// Mitsubishi GX Works2 project: project_PLC_Final   PLC: FX3G

// global labels: Global1
VAR_GLOBAL
  start_switch AT X007 : BOOL;
END_VAR
VAR_GLOBAL CONSTANT
  reset : REAL;
END_VAR
VAR_GLOBAL
  chocolate_stock AT D2000 : REAL;
  nuts_stock AT D2400 : REAL;
  pistachio_stock AT D2800 : REAL;
  kadaif_stock AT D3200 : REAL;
  chocolate_input AT D2200 : REAL;
  nuts_input AT D2600 : REAL;
  pistachio_input AT D3000 : REAL;
  kadaif_input AT D3400 : REAL;
END_VAR
VAR_GLOBAL CONSTANT
  melting_chocolate : REAL := 400;
  mix_nuts : REAL := 100;
  dubai_package : REAL := 120;
  mix_nuts_packge : REAL := 100;
  kadaif_dubai_package : REAL := 60;
END_VAR
VAR_GLOBAL
  m_28 AT M28 : BOOL;
  m_27 AT M27 : BOOL;
  m_26 AT M26 : BOOL;
  m_25 AT M25 : BOOL;
  m_29 AT M29 : BOOL;
  m_30 AT M30 : BOOL;
  m_31 AT M31 : BOOL;
  m_32 AT M32 : BOOL;
  valid_input AT M153 : BOOL;
  active_day AT Y007 : BOOL;
  end_day AT X005 : BOOL;
  start_melting AT X001 : BOOL;
  melting_container AT D4000 : REAL;
  m_0 AT M0 : BOOL;
  temp_sensor AT X002 : BOOL;
  melting_light AT Y001 : BOOL;
  location_sensor AT X003 : BOOL;
  casting_container AT D4200 : REAL;
  finish_casting AT TS1 : BOOL;
  casting_in_process AT Y002 : BOOL;
  casting AT TC1 : BOOL;
END_VAR
VAR_GLOBAL CONSTANT
  casting_time : INT := 40;
END_VAR
VAR_GLOBAL
  choosing_switch AT X004 : BOOL;
  analog_input AT D8280 : INT;
END_VAR
VAR_GLOBAL CONSTANT
  convert : REAL := 400;
END_VAR
VAR_GLOBAL
  analog_input1_sample AT M5 : BOOL;
  save_analog_input1 AT D4600 : REAL;
END_VAR
VAR_GLOBAL CONSTANT
  max5 : REAL := 5;
END_VAR
VAR_GLOBAL
  nuts_mix AT M2 : BOOL;
END_VAR
VAR_GLOBAL CONSTANT
  min5 : REAL := 5;
  max10 : REAL := 10;
END_VAR
VAR_GLOBAL
  dubai AT M1 : BOOL;
  analog_real AT D1200 : REAL;
  filling_container AT D4400 : REAL;
  ready_filling_mix AT M6 : BOOL;
END_VAR
VAR_GLOBAL CONSTANT
  mix_pistachio : REAL := 100;
  dubai_nuts : REAL := 20;
  dubai_pistachio : REAL := 120;
  dubai_kadaif : REAL := 60;
END_VAR
VAR_GLOBAL
  ready_filling_dubai AT M7 : BOOL;
  tc_2 AT TC2 : BOOL;
END_VAR
VAR_GLOBAL CONSTANT
  five_sec : INT := 50;
END_VAR
VAR_GLOBAL
  flashing_5_sec AT M100 : BOOL;
  m_105 AT M105 : BOOL;
  tc_3 AT TC3 : BOOL;
END_VAR
VAR_GLOBAL CONSTANT
  one_sec : INT := 10;
END_VAR
VAR_GLOBAL
  ts_3 AT TS3 : BOOL;
  y_3 AT Y003 : BOOL;
  ts_4 AT TS4 : BOOL;
  tc_4 AT TC4 : BOOL;
  y_4 AT Y004 : BOOL;
  ts_2 AT TS2 : BOOL;
  cooling_switch AT X006 : BOOL;
  cooling_container AT D5000 : REAL;
END_VAR
VAR_GLOBAL CONSTANT
  zero : INT;
END_VAR
VAR_GLOBAL
  tc_5 AT TC5 : BOOL;
END_VAR
VAR_GLOBAL CONSTANT
  sec_3 : INT := 30;
END_VAR
VAR_GLOBAL
  ts_5 AT TS5 : BOOL;
  cooling_light AT Y006 : BOOL;
  table_packing AT X000 : BOOL;
  package_counter AT CC1 : BOOL;
END_VAR
VAR_GLOBAL CONSTANT
  four_table : INT := 3;
END_VAR
VAR_GLOBAL
  package_count AT CS1 : BOOL;
  packing_light AT Y005 : BOOL;
  finish_packing AT M51 : BOOL;
END_VAR
VAR_GLOBAL CONSTANT
  package : INT := 4;
END_VAR
VAR_GLOBAL
  storage_container AT D7000 : REAL;
END_VAR
VAR_GLOBAL CONSTANT
  add_package : REAL := 1;
  converting_to_analog_output : REAL := 40;
END_VAR
VAR_GLOBAL
  analog_output AT D8282 : INT;
END_VAR

// task Task_01 (event TRUE, interval 0, priority 31): POU_01

PROGRAM POU_01
(* structured ladder/FBD written out as ST: instructions are called as NAME(EN, inputs, outputs); _pN, _eN, _tN stand for wires *)
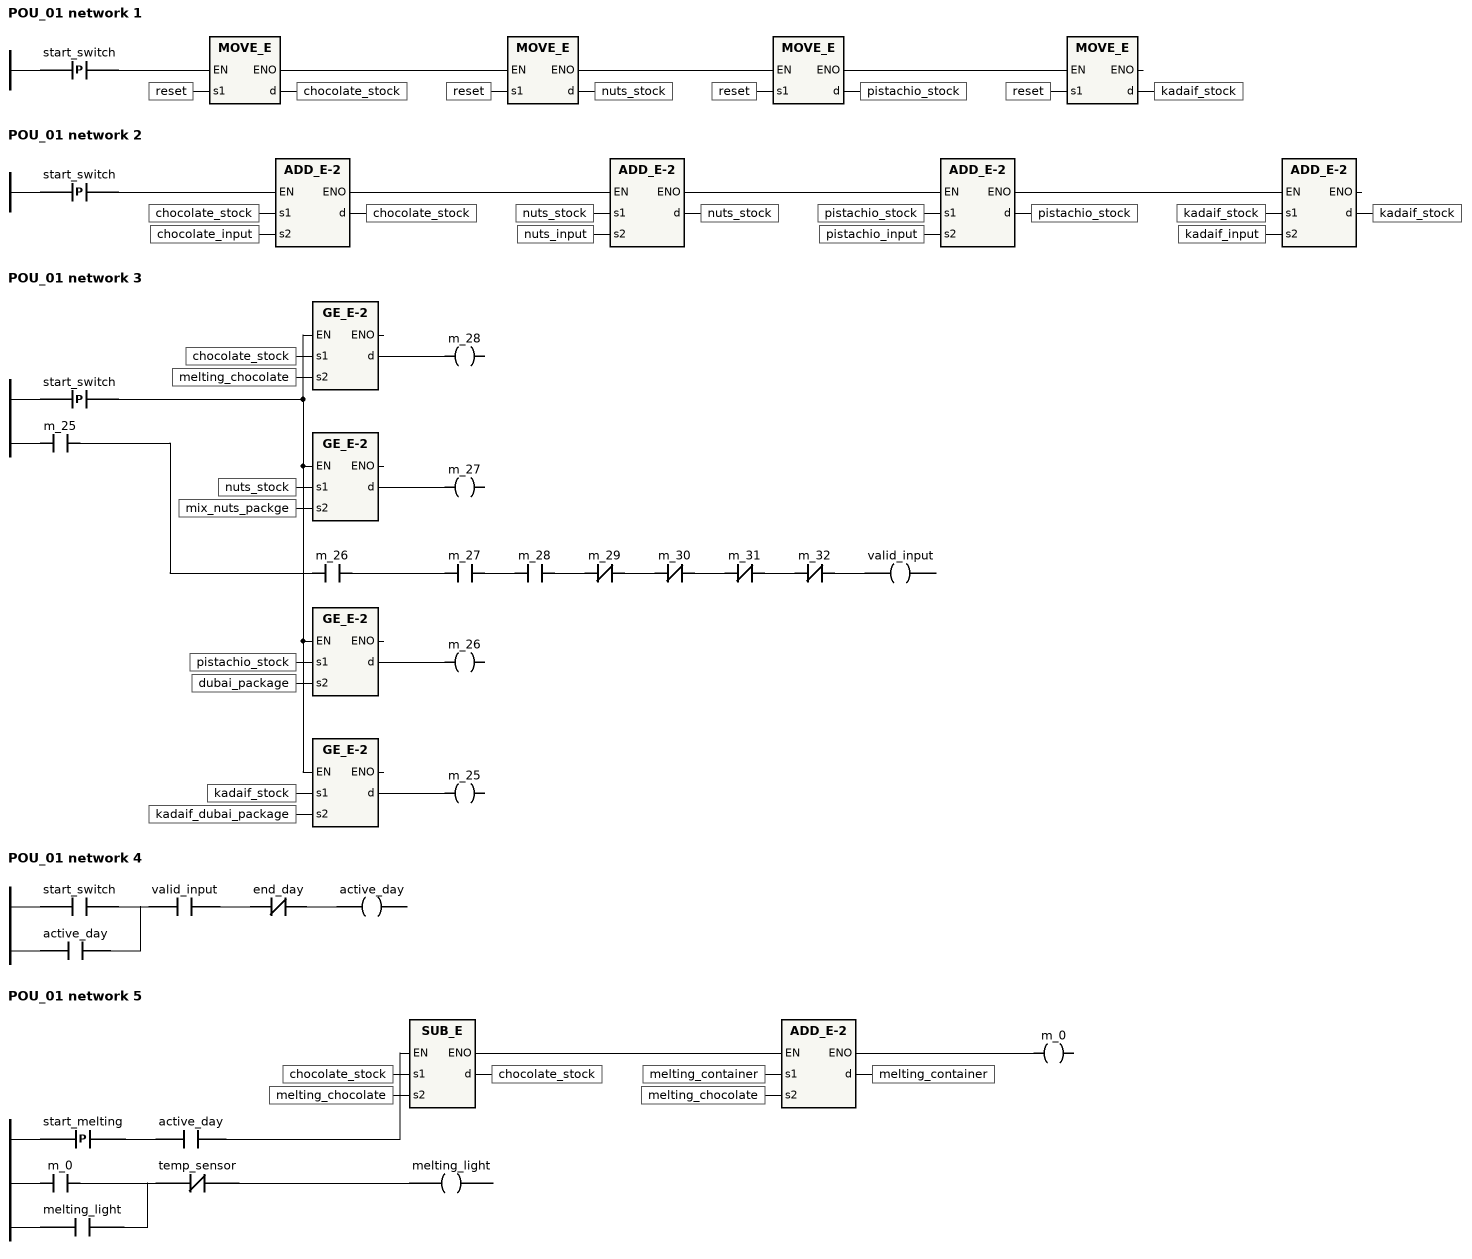
(* network 1 *)
_e1 := MOVE_E(LDP(TRUE, start_switch), reset, chocolate_stock);
_e2 := MOVE_E(_e1, reset, nuts_stock);
_e3 := MOVE_E(_e2, reset, pistachio_stock);
MOVE_E(_e3, reset, kadaif_stock);
(* network 2 *)
_e1 := ADD_E(LDP(TRUE, start_switch), chocolate_stock, chocolate_input, chocolate_stock);
_e2 := ADD_E(_e1, nuts_stock, nuts_input, nuts_stock);
_e3 := ADD_E(_e2, pistachio_stock, pistachio_input, pistachio_stock);
ADD_E(_e3, kadaif_stock, kadaif_input, kadaif_stock);
(* network 3 *)
_p1 := LDP(TRUE, start_switch);
GE_E(_p1, chocolate_stock, melting_chocolate, _t2);
m_28 := _t2;
GE_E(_p1, nuts_stock, mix_nuts_packge, _t3);
m_27 := _t3;
GE_E(_p1, pistachio_stock, dubai_package, _t4);
m_26 := _t4;
GE_E(_p1, kadaif_stock, kadaif_dubai_package, _t5);
m_25 := _t5;
valid_input := m_25 AND m_26 AND m_27 AND m_28 AND NOT m_29 AND NOT m_30 AND NOT m_31 AND NOT m_32;
(* network 4 *)
active_day := ((start_switch OR active_day) AND valid_input) AND NOT end_day;
(* network 5 *)
_e1 := SUB_E(LDP(TRUE, start_melting) AND active_day, chocolate_stock, melting_chocolate, chocolate_stock);
_e2 := ADD_E(_e1, melting_container, melting_chocolate, melting_container);
m_0 := _e2;
melting_light := (m_0 OR melting_light) AND NOT temp_sensor;
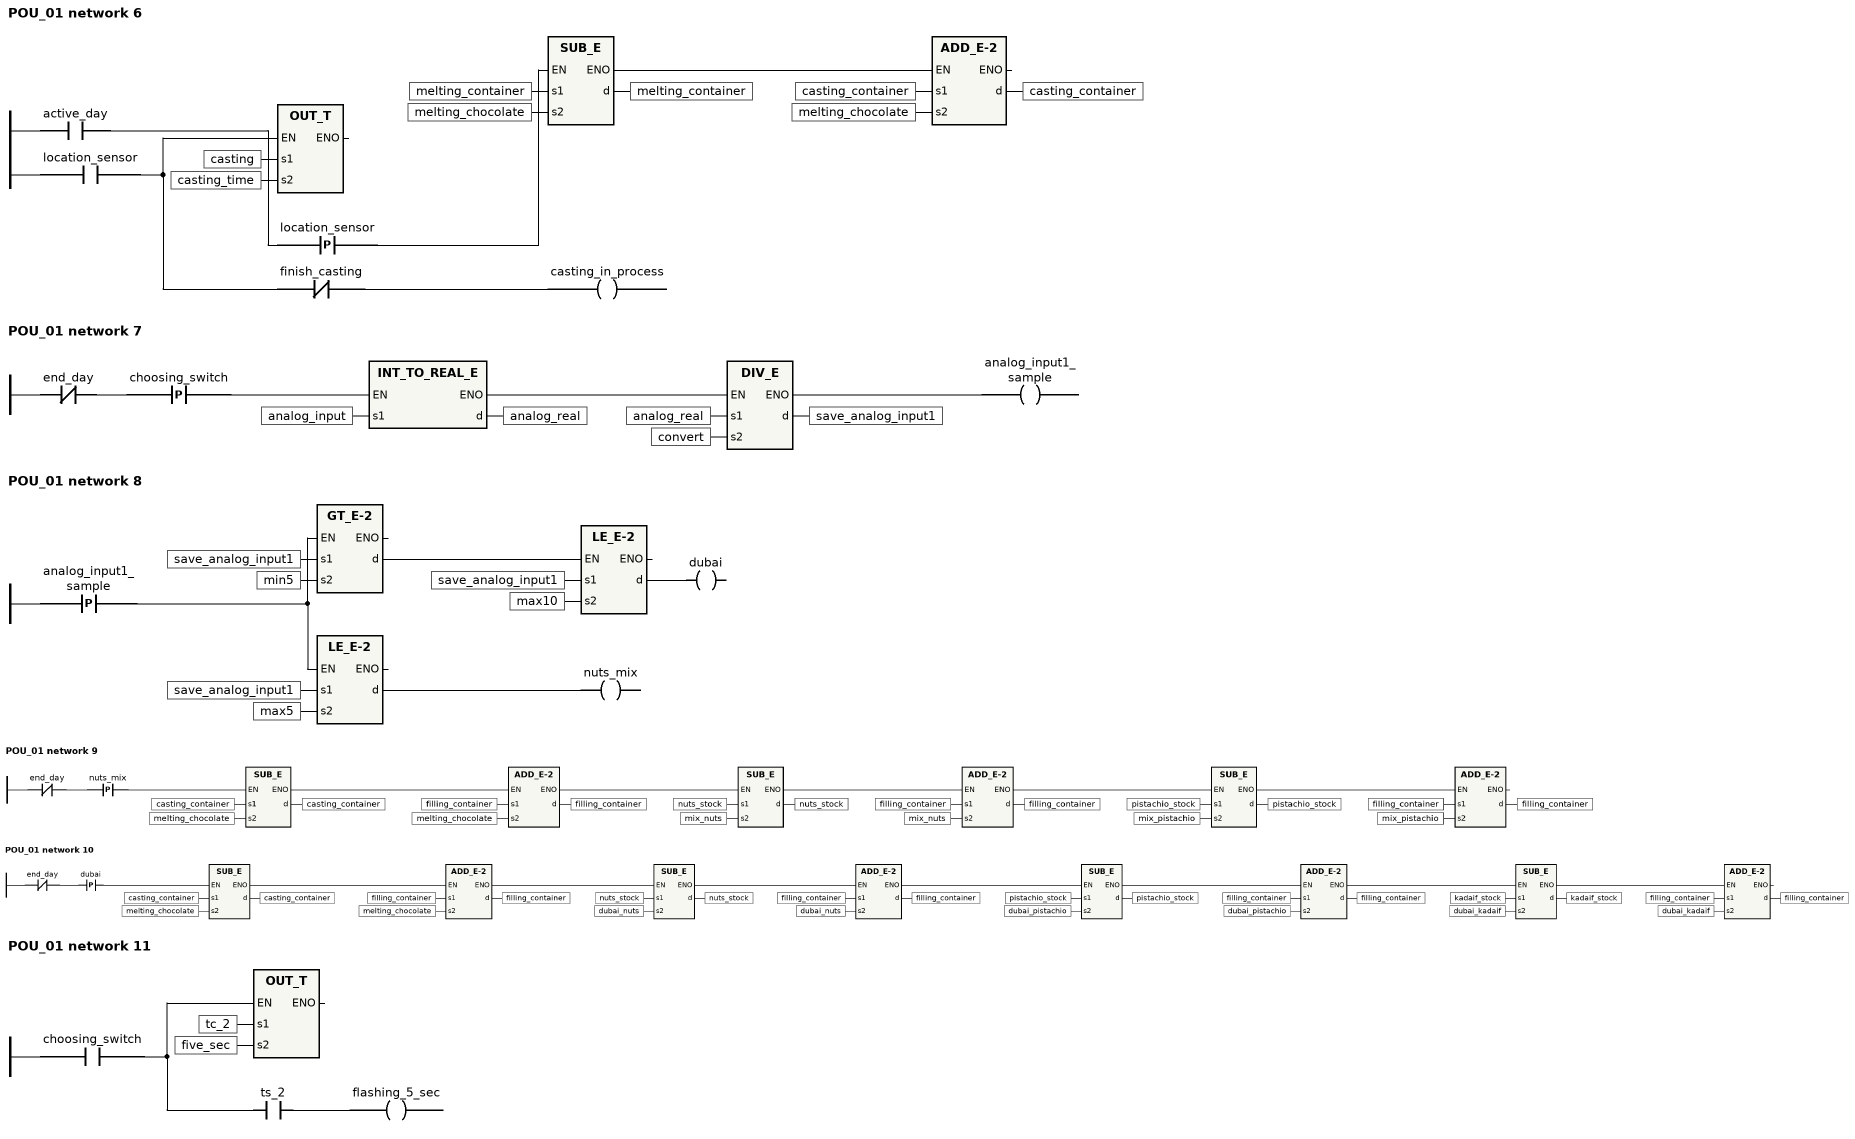
(* network 6 *)
_e1 := SUB_E(active_day AND LDP(TRUE, location_sensor), melting_container, melting_chocolate, melting_container);
ADD_E(_e1, casting_container, melting_chocolate, casting_container);
OUT_T(location_sensor, casting, casting_time);
casting_in_process := location_sensor AND NOT finish_casting;
(* network 7 *)
_e1 := INT_TO_REAL_E(NOT end_day AND LDP(TRUE, choosing_switch), analog_input, analog_real);
_e2 := DIV_E(_e1, analog_real, convert, save_analog_input1);
analog_input1_sample := _e2;
(* network 8 *)
_p1 := LDP(TRUE, analog_input1_sample);
LE_E(_p1, save_analog_input1, max5, _t2);
nuts_mix := _t2;
GT_E(_p1, save_analog_input1, min5, _t3);
LE_E(_t3, save_analog_input1, max10, _t4);
dubai := _t4;
(* network 9 *)
_e1 := SUB_E(NOT end_day AND LDP(TRUE, nuts_mix), casting_container, melting_chocolate, casting_container);
_e2 := ADD_E(_e1, filling_container, melting_chocolate, filling_container);
_e3 := SUB_E(_e2, nuts_stock, mix_nuts, nuts_stock);
_e4 := ADD_E(_e3, filling_container, mix_nuts, filling_container);
_e5 := SUB_E(_e4, pistachio_stock, mix_pistachio, pistachio_stock);
ADD_E(_e5, filling_container, mix_pistachio, filling_container);
(* network 10 *)
_e1 := SUB_E(NOT end_day AND LDP(TRUE, dubai), casting_container, melting_chocolate, casting_container);
_e2 := ADD_E(_e1, filling_container, melting_chocolate, filling_container);
_e3 := SUB_E(_e2, nuts_stock, dubai_nuts, nuts_stock);
_e4 := ADD_E(_e3, filling_container, dubai_nuts, filling_container);
_e5 := SUB_E(_e4, pistachio_stock, dubai_pistachio, pistachio_stock);
_e6 := ADD_E(_e5, filling_container, dubai_pistachio, filling_container);
_e7 := SUB_E(_e6, kadaif_stock, dubai_kadaif, kadaif_stock);
ADD_E(_e7, filling_container, dubai_kadaif, filling_container);
(* network 11 *)
OUT_T(choosing_switch, tc_2, five_sec);
flashing_5_sec := choosing_switch AND ts_2;
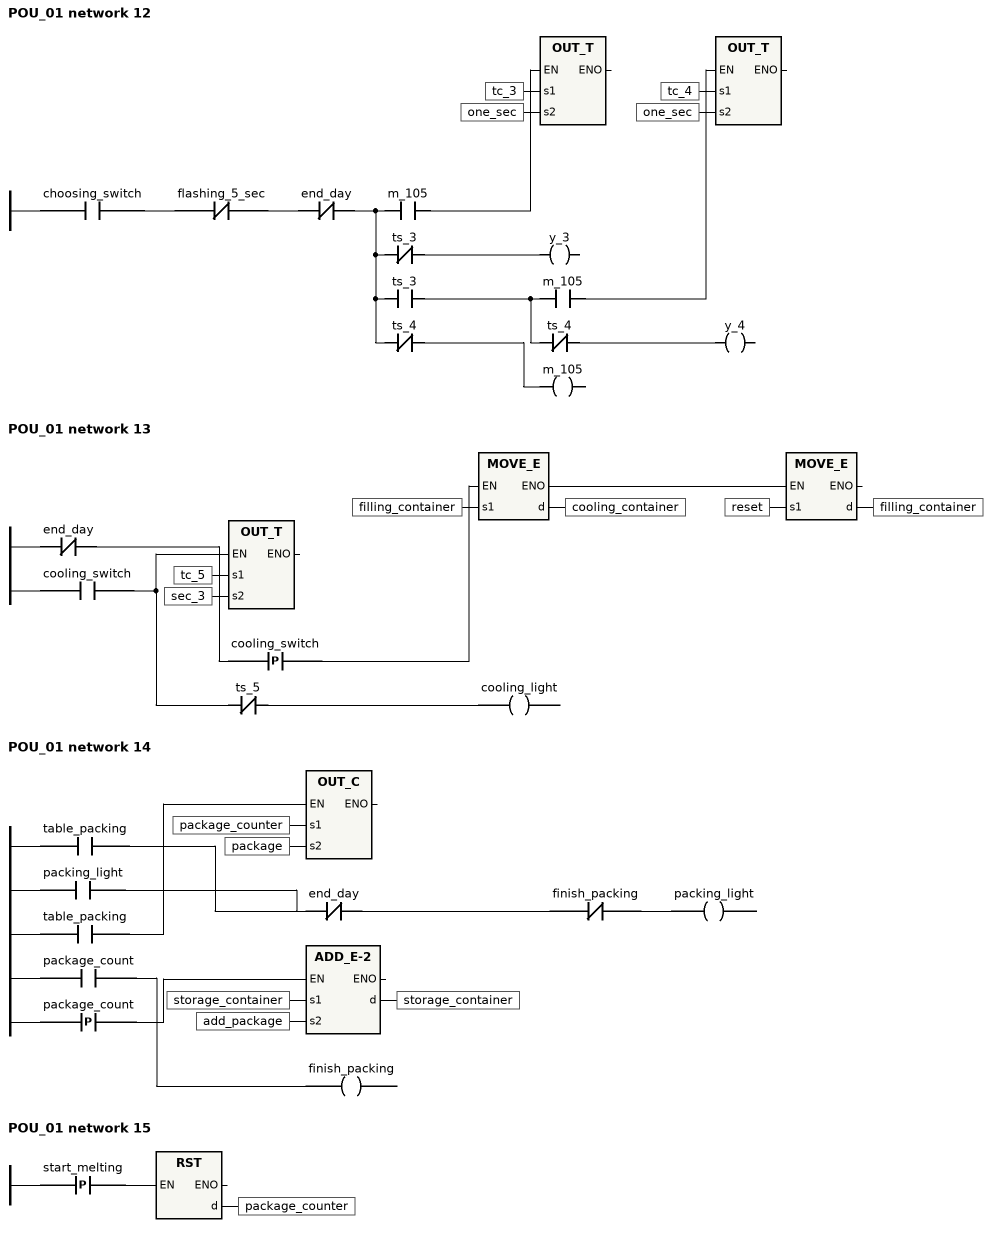
(* network 12 *)
_p1 := choosing_switch AND NOT flashing_5_sec AND NOT end_day;
OUT_T(_p1 AND m_105, tc_3, one_sec);
y_3 := _p1 AND NOT ts_3;
_p2 := _p1 AND ts_3;
OUT_T(_p2 AND m_105, tc_4, one_sec);
y_4 := _p2 AND NOT ts_4;
m_105 := _p1 AND NOT ts_4;
(* network 13 *)
_e1 := MOVE_E(NOT end_day AND LDP(TRUE, cooling_switch), filling_container, cooling_container);
MOVE_E(_e1, reset, filling_container);
OUT_T(cooling_switch, tc_5, sec_3);
cooling_light := cooling_switch AND NOT ts_5;
(* network 14 *)
packing_light := ((table_packing OR packing_light) AND NOT end_day) AND NOT finish_packing;
OUT_C(table_packing, package_counter, package);
finish_packing := package_count;
ADD_E(LDP(TRUE, package_count), storage_container, add_package, storage_container);
(* network 15 *)
RST(LDP(TRUE, start_melting), package_counter);
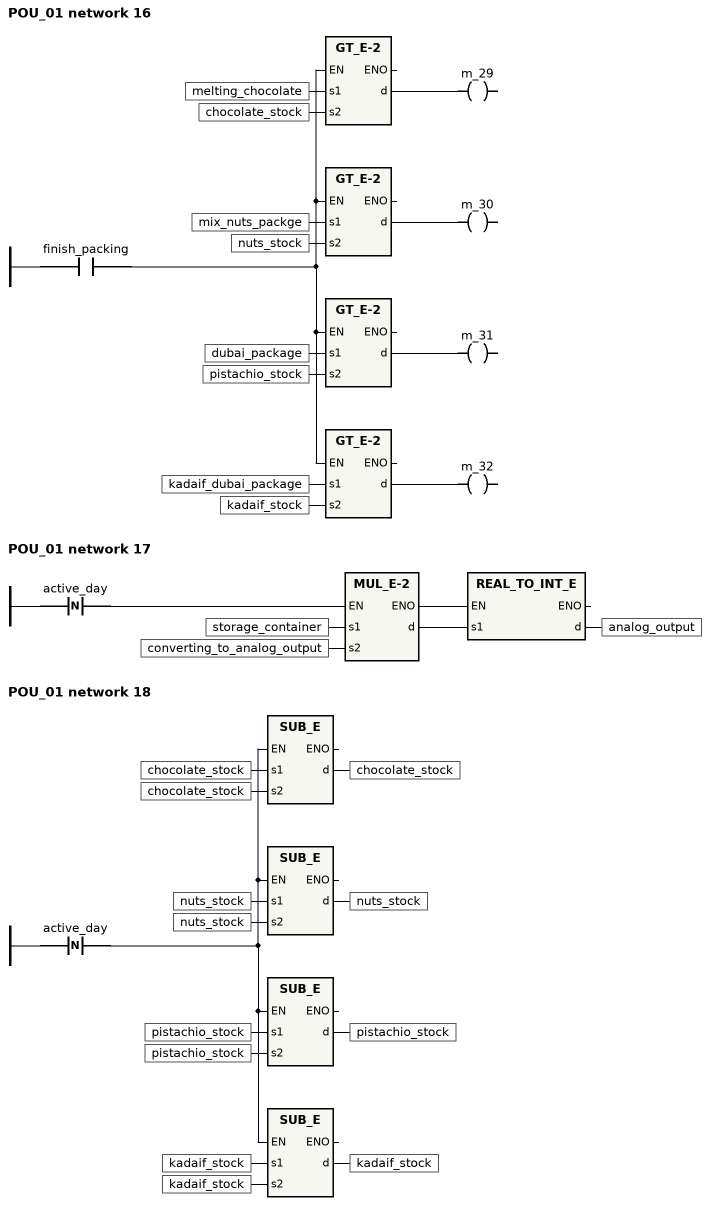
(* network 16 *)
GT_E(finish_packing, melting_chocolate, chocolate_stock, _t1);
m_29 := _t1;
GT_E(finish_packing, mix_nuts_packge, nuts_stock, _t2);
m_30 := _t2;
GT_E(finish_packing, dubai_package, pistachio_stock, _t3);
m_31 := _t3;
GT_E(finish_packing, kadaif_dubai_package, kadaif_stock, _t4);
m_32 := _t4;
(* network 17 *)
_e2 := MUL_E(LDF(TRUE, active_day), storage_container, converting_to_analog_output, _t1);
REAL_TO_INT_E(_e2, _t1, analog_output);
(* network 18 *)
_p1 := LDF(TRUE, active_day);
SUB_E(_p1, chocolate_stock, chocolate_stock, chocolate_stock);
SUB_E(_p1, nuts_stock, nuts_stock, nuts_stock);
SUB_E(_p1, pistachio_stock, pistachio_stock, pistachio_stock);
SUB_E(_p1, kadaif_stock, kadaif_stock, kadaif_stock);
END_PROGRAM
